FUNCTION_BLOCK DigitalInput_NO_TEST
VAR
END_VAR

ForcedOn();
ForcedOff();
On();
Off();

METHOD ForcedOff : BOOL
VAR
	Expected		: BOOL;
	Actual			: BOOL;
	Input			: BOOL;
	DigitalInput_NO : DigitalInput_NO('DigitalInput', Input);
END_VAR
IF TestSuite.Test(__POUNAME()).ExecuteTest() THEN
	Expected			  := FALSE;
	DigitalInput_NO.Force := E_ForceState.ForceOff;
	Input				  := TRUE;
	Actual				  := DigitalInput_NO.IsActive;
	TestSuite.Test(__POUNAME()).AssertEqual(Expected, Actual);
END_IF
END_METHOD

METHOD ForcedOn : BOOL
VAR
	Expected		: BOOL;
	Actual			: BOOL;
	Input			: BOOL;
	DigitalInput_NO : DigitalInput_NO('DigitalInput', Input);
END_VAR
IF TestSuite.Test(__POUNAME()).ExecuteTest() THEN
	Expected			  := TRUE;
	DigitalInput_NO.Force := E_ForceState.ForceOn;
	Input				  := FALSE;
	Actual				  := DigitalInput_NO.IsActive;
	TestSuite.Test(__POUNAME()).AssertEqual(Expected, Actual);
END_IF
END_METHOD

METHOD Off : BOOL
VAR
	Expected		: BOOL;
	Actual			: BOOL;
	Input			: BOOL;
	DigitalInput_NO : DigitalInput_NO('DigitalInput', Input);
END_VAR
IF TestSuite.Test(__POUNAME()).ExecuteTest() THEN
	Expected			  := FALSE;
	DigitalInput_NO.Force := E_ForceState.Unforced;
	Input				  := FALSE;
	Actual				  := DigitalInput_NO.IsActive;
	TestSuite.Test(__POUNAME()).AssertEqual(Expected, Actual);
END_IF
END_METHOD

METHOD On
VAR
	Expected		: BOOL;
	Actual			: BOOL;
	Input			: BOOL;
	DigitalInput_NO : DigitalInput_NO('DigitalInput', Input);
END_VAR
IF TestSuite.Test(__POUNAME()).ExecuteTest() THEN
	Expected			  := TRUE;
	DigitalInput_NO.Force := E_ForceState.Unforced;
	Input				  := TRUE;
	Actual				  := DigitalInput_NO.IsActive;
	TestSuite.Test(__POUNAME()).AssertEqual(Expected, Actual);
END_IF
END_METHOD

END_FUNCTION_BLOCK

(* stored: Version 1.1.0.1, ProductVersion 3.1.4026.18
   POU DigitalInput_NO_TEST: Id {f9f73e65-4f99-43b7-b834-6ebbd09ac1c5}, SpecialFunc None
   Method ForcedOff: Id {0cb60847-7184-49f1-82d2-202a9cc563fe}
   Method ForcedOn: Id {5a0e859f-90b7-4cfd-b965-c80735e0acf0}
   Method Off: Id {b782b061-1052-4095-8de0-f1324df7bc8c}
   Method On: Id {f7828c4c-27e4-4bf5-b5c6-53c6b2dd52d9} *)
